// Mitsubishi GX Works2 project: PLC_GROUP2_Final   PLC: FX3G

// global labels: Global1
VAR_GLOBAL
  StartDay AT X007 : BOOL;
  StartRaspberryStock AT D1101 : REAL;
  StartLemonStock AT D1103 : REAL;
  StartStabilizerStock AT D1105 : REAL;
  StartGummyBearsStock AT D1107 : REAL;
  StockRaspberry AT D1111 : REAL;
  LemonStock AT D1133 : REAL;
  RaspberryStock AT D1111 : REAL;
  StabilizerStock AT D1155 : REAL;
  GummyBearsStock AT D1177 : REAL;
  WorkDayLight AT Y007 : BOOL;
  LackOfStock AT M0 : BOOL;
  EmergencySwitch AT X005 : BOOL;
  WorkDayLigth AT Y007 : BOOL;
  IceCreamFlavors AT X001 : BOOL;
  AnalogInput1 AT D8280 : INT;
  SaveAnalogInput1 AT D8201 : INT;
  Analog1AsFloat AT D1221 : REAL;
  Divider AT E400 : REAL;
  IndicatorLigth AT M1 : BOOL;
  RegularLigth AT M2 : BOOL;
  IndulgenceLigth AT M3 : BOOL;
  CheckStock AT M100 : BOOL;
END_VAR
VAR_GLOBAL CONSTANT
  RaspberryForPackage : REAL := 280;
END_VAR
VAR_GLOBAL
  RegularPackage AT M22 : BOOL;
END_VAR
VAR_GLOBAL CONSTANT
  Regular : REAL := 5;
END_VAR
VAR_GLOBAL
  RegularCheck AT M2 : BOOL;
  IndulgencePackage AT M33 : BOOL;
END_VAR
VAR_GLOBAL CONSTANT
  Indulgence : INT := 6;
  IndulgenceMin : REAL := 6;
  LemonForPackage : REAL := 455;
  StabilizerForPackage : REAL := 105;
  GummyBearsForPackage : REAL := 28;
  RaspberryForPackage3 : REAL := 385;
  LemonForPackage3 : REAL := 665;
  StabilizerForPackage3 : REAL := 210;
  GummyBearsForPackage3 : REAL := 70;
  RaspberryForPackage2 : INT := 280;
  GummyBearsForPackage2 : INT := 280;
  addRaspberry : REAL := 350;
  addLemon : REAL := 490;
  addRaspberry3 : REAL := 560;
  addLemon3 : REAL := 700;
END_VAR
VAR_GLOBAL
  FlavorsMaking AT M40 : BOOL;
END_VAR
VAR_GLOBAL CONSTANT
  TotIceCreamTime : INT := 50;
END_VAR
VAR_GLOBAL
  IceCreamTime AT TC1 : BOOL;
  MakingTime AT Y000 : BOOL;
  MakingTimer AT TS1 : BOOL;
  Cooling AT X002 : BOOL;
  TemperatureSensor AT X003 : BOOL;
END_VAR
VAR_GLOBAL CONSTANT
  MaxTime : INT := 80;
END_VAR
VAR_GLOBAL
  CoolingTime AT TC8 : BOOL;
  CoolingTimer AT TS8 : BOOL;
  CoolingLight AT Y002 : BOOL;
END_VAR
VAR_GLOBAL CONSTANT
  GummyBearskForPackage : REAL := 28;
  GummyBearskForPackage3 : REAL := 70;
END_VAR
VAR_GLOBAL
  RegularMix AT M4 : BOOL;
  IndulgenceMix AT M5 : BOOL;
END_VAR
VAR_GLOBAL CONSTANT
  RegularMix3sec : INT := 30;
  IndulgenceMix5sec : INT := 50;
END_VAR
VAR_GLOBAL
  StartMix AT M4 : BOOL;
  LightTimer AT TS9 : BOOL;
  LightTime AT TC9 : BOOL;
  FirstLight AT Y005 : BOOL;
  SecondLight AT Y006 : BOOL;
  HelpLight AT M5 : BOOL;
  FirstLightTime AT TC10 : BOOL;
  SecondLightTime AT TC11 : BOOL;
  FirstLightTimer AT TS10 : BOOL;
  SecondLightTimer AT TS11 : BOOL;
  IndulgenceChecking AT M6 : BOOL;
  CoolingRaspberry AT D2004 : REAL;
  CoolingLemon AT D2006 : REAL;
  MixingFlavors AT D3000 : REAL;
END_VAR
VAR_GLOBAL CONSTANT
  Restart : INT;
END_VAR
VAR_GLOBAL
  AnalogOutput AT D8282 : INT;
  RaspberryIceCream AT D2000 : REAL;
  LemonIceCream AT D2002 : REAL;
  Checking AT Y010 : BOOL;
  ch AT Y011 : BOOL;
  StayOn AT M50 : BOOL;
  Help AT M50 : BOOL;
  FlavorsMaking12 AT M42 : BOOL;
  HelpCooling AT M60 : BOOL;
  MixTimerWord AT D3006 : INT;
  MixTimer AT D3002 : REAL;
END_VAR
VAR_GLOBAL CONSTANT
  MaxTime2 : INT := 8;
END_VAR
VAR_GLOBAL
  LightTime3 AT TC12 : BOOL;
  LightTimer3 AT TS12 : BOOL;
  Help7 AT M7 : BOOL;
  Check4 AT Y010 : BOOL;
  Check10 AT Y004 : BOOL;
  Packing AT X004 : BOOL;
END_VAR
VAR_GLOBAL CONSTANT
  RstMixingFlavors : REAL;
END_VAR
VAR_GLOBAL
  OneCone AT X000 : BOOL;
  FirstConeCounter AT CC0 : BOOL;
END_VAR
VAR_GLOBAL CONSTANT
  FirstCone : INT := 1;
END_VAR
VAR_GLOBAL
  ConesCounter AT CC1 : BOOL;
END_VAR
VAR_GLOBAL CONSTANT
  SevenCones : INT := 7;
END_VAR
VAR_GLOBAL
  AfterFirstCone AT CS0 : BOOL;
  FinishPackeg AT CS1 : BOOL;
  FinishPackage AT CS1 : BOOL;
  PackingLigth AT Y004 : BOOL;
END_VAR
VAR_GLOBAL CONSTANT
  NewPackage : REAL := 1;
END_VAR
VAR_GLOBAL
  TotalPackages AT D5555 : REAL;
END_VAR
VAR_GLOBAL CONSTANT
  Mult : REAL := 40;
  Reset : REAL;
END_VAR
VAR_GLOBAL
  StartReset AT M8 : BOOL;
  HelpM41 AT M41 : BOOL;
  closeLigth AT M100 : BOOL;
END_VAR

// task Task_01 (event TRUE, interval 0, priority 31): POU_01

PROGRAM POU_01
(* structured ladder/FBD written out as ST: instructions are called as NAME(EN, inputs, outputs); _pN, _eN, _tN stand for wires *)
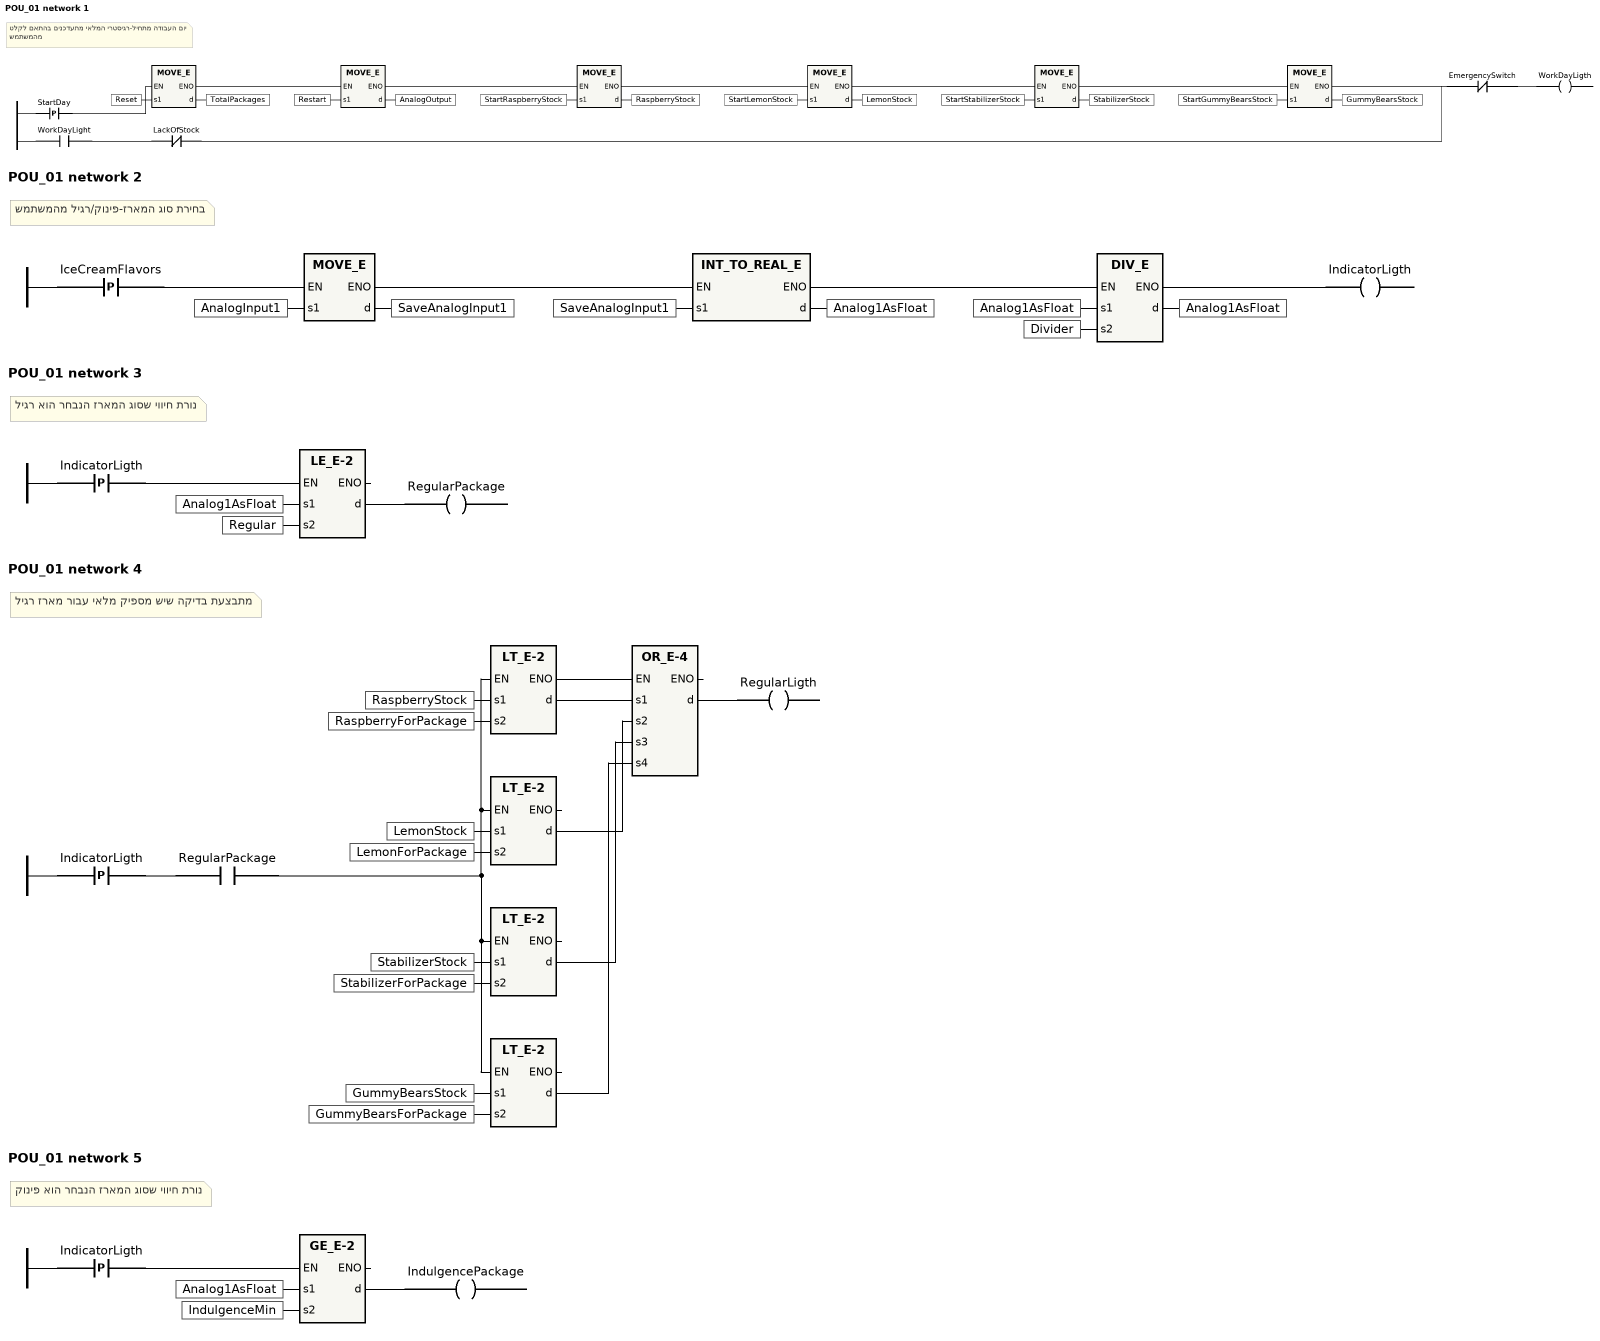
(* network 1 Start workday *)
(* יום העבודה מתחיל-רגיסטרי המלאי מתעדכנים בהתאם לקלט מהמשתמש *)
_e1 := MOVE_E(LDP(TRUE, StartDay), Reset, TotalPackages);
_e2 := MOVE_E(_e1, Restart, AnalogOutput);
_e3 := MOVE_E(_e2, StartRaspberryStock, RaspberryStock);
_e4 := MOVE_E(_e3, StartLemonStock, LemonStock);
_e5 := MOVE_E(_e4, StartStabilizerStock, StabilizerStock);
_e6 := MOVE_E(_e5, StartGummyBearsStock, GummyBearsStock);
WorkDayLigth := (_e6 OR (WorkDayLight AND NOT LackOfStock)) AND NOT EmergencySwitch;
(* network 2 Type sampeling *)
(* בחירת סוג המארז-פינוק/רגיל מהמשתמש *)
_e1 := MOVE_E(LDP(TRUE, IceCreamFlavors), AnalogInput1, SaveAnalogInput1);
_e2 := INT_TO_REAL_E(_e1, SaveAnalogInput1, Analog1AsFloat);
_e3 := DIV_E(_e2, Analog1AsFloat, Divider, Analog1AsFloat);
IndicatorLigth := _e3;
(* network 3 If regular *)
(* נורת חיווי שסוג המארז הנבחר הוא רגיל *)
LE_E(LDP(TRUE, IndicatorLigth), Analog1AsFloat, Regular, _t1);
RegularPackage := _t1;
(* network 4 Check stock for R *)
(* מתבצעת בדיקה שיש מספיק מלאי עבור מארז רגיל *)
_p1 := LDP(TRUE, IndicatorLigth) AND RegularPackage;
_e3 := LT_E(_p1, RaspberryStock, RaspberryForPackage, _t2);
LT_E(_p1, LemonStock, LemonForPackage, _t4);
LT_E(_p1, StabilizerStock, StabilizerForPackage, _t5);
LT_E(_p1, GummyBearsStock, GummyBearsForPackage, _t6);
OR_E(_e3, _t2, _t4, _t5, _t6, _t7);
RegularLigth := _t7;
(* network 5 If indulgence *)
(* נורת חיווי שסוג המארז הנבחר הוא פינוק *)
GE_E(LDP(TRUE, IndicatorLigth), Analog1AsFloat, IndulgenceMin, _t1);
IndulgencePackage := _t1;
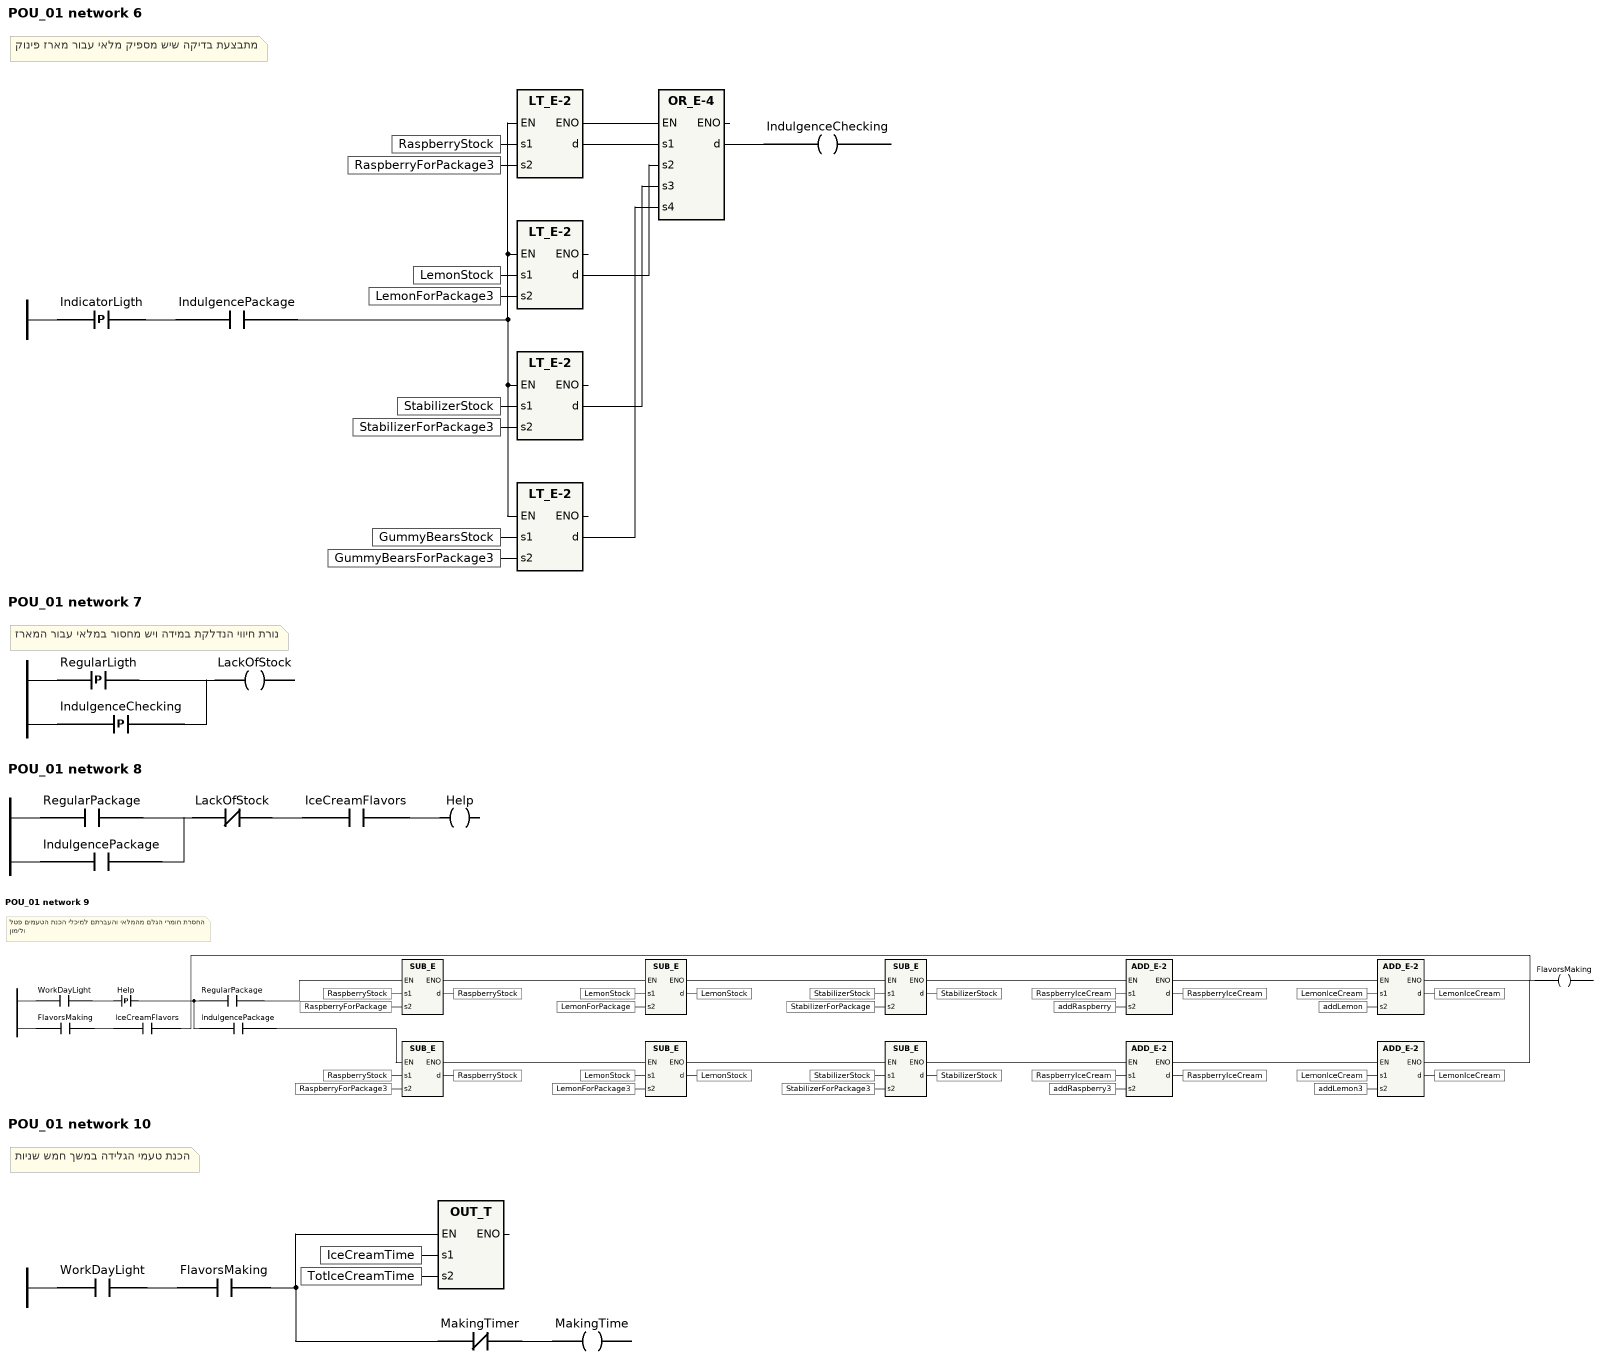
(* network 6 Check stock for I *)
(* מתבצעת בדיקה שיש מספיק מלאי עבור מארז פינוק *)
_p1 := LDP(TRUE, IndicatorLigth) AND IndulgencePackage;
_e3 := LT_E(_p1, RaspberryStock, RaspberryForPackage3, _t2);
LT_E(_p1, LemonStock, LemonForPackage3, _t4);
LT_E(_p1, StabilizerStock, StabilizerForPackage3, _t5);
LT_E(_p1, GummyBearsStock, GummyBearsForPackage3, _t6);
OR_E(_e3, _t2, _t4, _t5, _t6, _t7);
IndulgenceChecking := _t7;
(* network 7 Out of stock *)
(* נורת חיווי הנדלקת במידה ויש מחסור במלאי עבור המארז *)
LackOfStock := LDP(TRUE, RegularLigth) OR LDP(TRUE, IndulgenceChecking);
(* network 8 Checks conditions *)
Help := ((RegularPackage OR IndulgencePackage) AND NOT LackOfStock) AND IceCreamFlavors;
(* network 9 Sub stocks *)
(* החסרת חומרי הגלם מהמלאי והעברתם למיכלי הכנת הטעמים פטל ולימון *)
_p1 := WorkDayLight AND LDP(TRUE, Help);
_e2 := SUB_E(_p1 AND RegularPackage, RaspberryStock, RaspberryForPackage, RaspberryStock);
_e3 := SUB_E(_e2, LemonStock, LemonForPackage, LemonStock);
_e4 := SUB_E(_e3, StabilizerStock, StabilizerForPackage, StabilizerStock);
_e5 := ADD_E(_e4, RaspberryIceCream, addRaspberry, RaspberryIceCream);
_e6 := ADD_E(_e5, LemonIceCream, addLemon, LemonIceCream);
_e7 := SUB_E(_p1 AND IndulgencePackage, RaspberryStock, RaspberryForPackage3, RaspberryStock);
_e8 := SUB_E(_e7, LemonStock, LemonForPackage3, LemonStock);
_e9 := SUB_E(_e8, StabilizerStock, StabilizerForPackage3, StabilizerStock);
_e10 := ADD_E(_e9, RaspberryIceCream, addRaspberry3, RaspberryIceCream);
_e11 := ADD_E(_e10, LemonIceCream, addLemon3, LemonIceCream);
FlavorsMaking := _e6 OR _e11 OR (FlavorsMaking AND IceCreamFlavors);
(* network 10 Flavors Making *)
(* הכנת טעמי הגלידה במשך חמש שניות *)
_p1 := WorkDayLight AND FlavorsMaking;
OUT_T(_p1, IceCreamTime, TotIceCreamTime);
MakingTime := _p1 AND NOT MakingTimer;
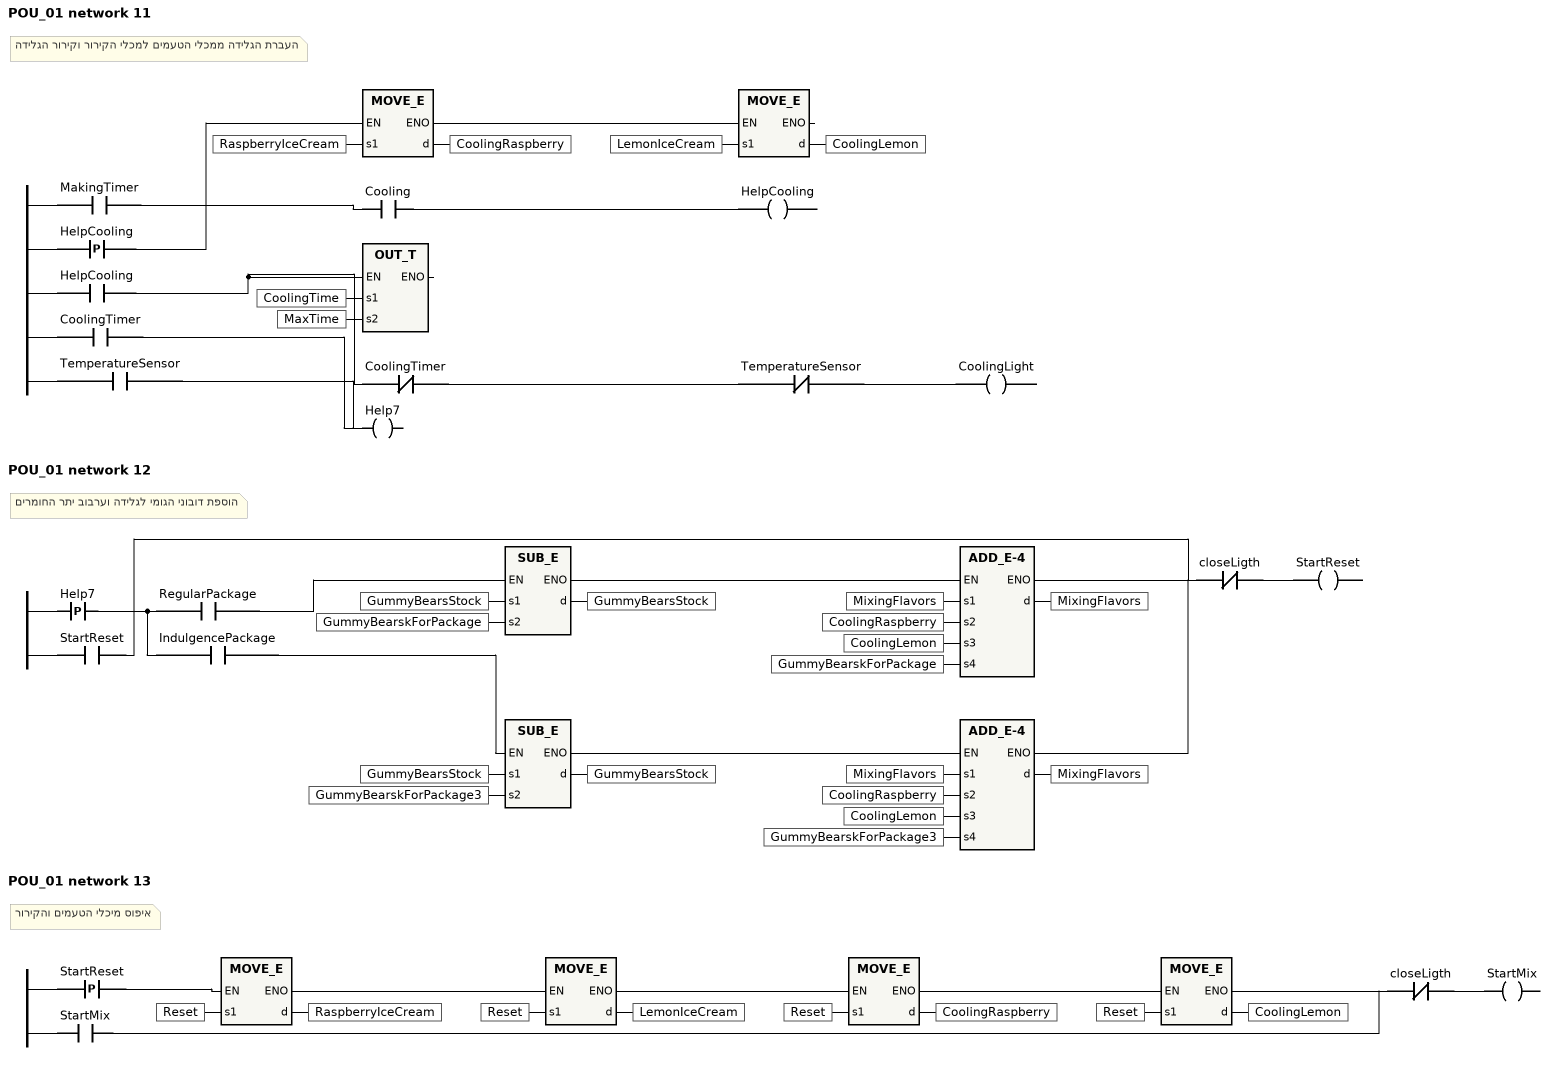
(* network 11 Cooling phase *)
(* העברת הגלידה ממכלי הטעמים למכלי הקירור וקירור הגלידה *)
HelpCooling := MakingTimer AND Cooling;
_e1 := MOVE_E(LDP(TRUE, HelpCooling), RaspberryIceCream, CoolingRaspberry);
MOVE_E(_e1, LemonIceCream, CoolingLemon);
OUT_T(HelpCooling, CoolingTime, MaxTime);
CoolingLight := HelpCooling AND NOT CoolingTimer AND NOT TemperatureSensor;
Help7 := CoolingTimer OR TemperatureSensor;
(* network 12 Prepar to Mixing *)
(* הוספת דובוני הגומי לגלידה וערבוב יתר החומרים *)
_p1 := LDP(TRUE, Help7);
_e2 := SUB_E(_p1 AND RegularPackage, GummyBearsStock, GummyBearskForPackage, GummyBearsStock);
_e3 := ADD_E(_e2, MixingFlavors, CoolingRaspberry, CoolingLemon, GummyBearskForPackage, MixingFlavors);
_e4 := SUB_E(_p1 AND IndulgencePackage, GummyBearsStock, GummyBearskForPackage3, GummyBearsStock);
_e5 := ADD_E(_e4, MixingFlavors, CoolingRaspberry, CoolingLemon, GummyBearskForPackage3, MixingFlavors);
StartReset := (_e3 OR _e5 OR StartReset) AND NOT closeLigth;
(* network 13 Restart *)
(* איפוס מיכלי הטעמים והקירור *)
_e1 := MOVE_E(LDP(TRUE, StartReset), Reset, RaspberryIceCream);
_e2 := MOVE_E(_e1, Reset, LemonIceCream);
_e3 := MOVE_E(_e2, Reset, CoolingRaspberry);
_e4 := MOVE_E(_e3, Reset, CoolingLemon);
StartMix := (_e4 OR StartMix) AND NOT closeLigth;
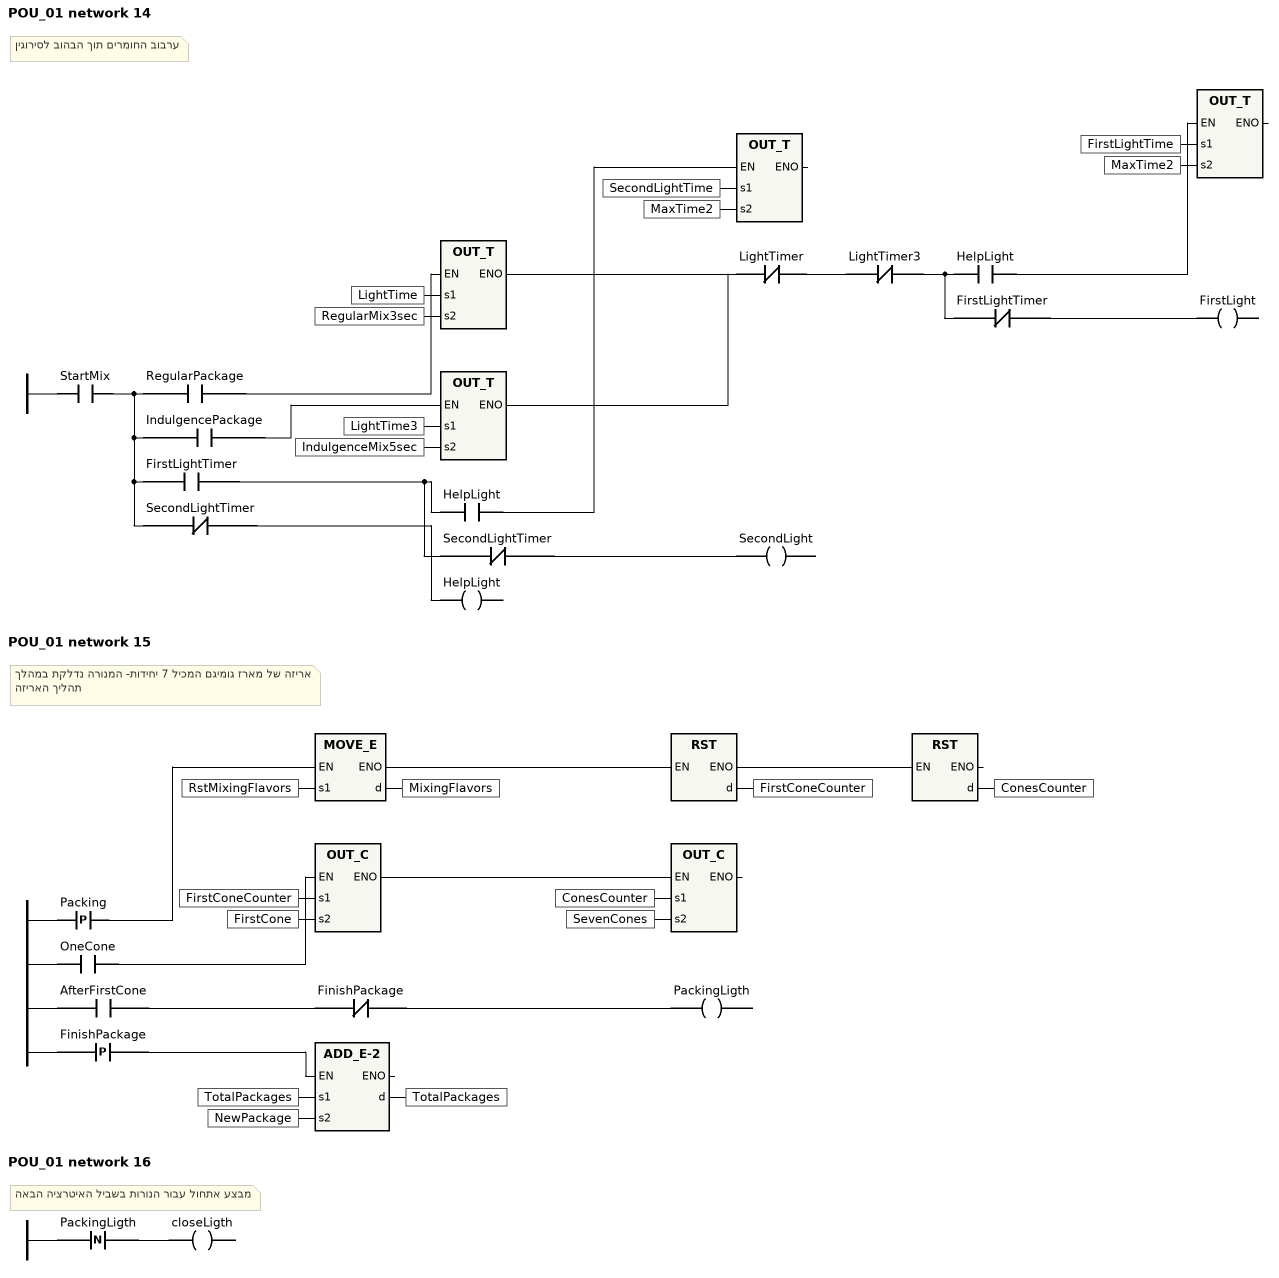
(* network 14 Mixing Ingredients *)
(* ערבוב החומרים תוך הבהוב לסירוגין *)
_e1 := OUT_T(StartMix AND RegularPackage, LightTime, RegularMix3sec);
_e2 := OUT_T(StartMix AND IndulgencePackage, LightTime3, IndulgenceMix5sec);
_p3 := ((_e1 OR _e2) AND NOT LightTimer) AND NOT LightTimer3;
OUT_T(_p3 AND HelpLight, FirstLightTime, MaxTime2);
FirstLight := _p3 AND NOT FirstLightTimer;
_p4 := StartMix AND FirstLightTimer;
OUT_T(_p4 AND HelpLight, SecondLightTime, MaxTime2);
SecondLight := _p4 AND NOT SecondLightTimer;
HelpLight := StartMix AND NOT SecondLightTimer;
(* network 15 Packing cones *)
(* אריזה של מארז גומיגם המכיל 7 יחידות- המנורה נדלקת במהלך תהליך האריזה *)
_e1 := MOVE_E(LDP(TRUE, Packing), RstMixingFlavors, MixingFlavors);
_e2 := RST(_e1, FirstConeCounter);
RST(_e2, ConesCounter);
_e3 := OUT_C(OneCone, FirstConeCounter, FirstCone);
OUT_C(_e3, ConesCounter, SevenCones);
PackingLigth := AfterFirstCone AND NOT FinishPackage;
ADD_E(LDP(TRUE, FinishPackage), TotalPackages, NewPackage, TotalPackages);
(* network 16 Restart bulbs *)
(* מבצע אתחול עבור הנורות בשביל האיטרציה הבאה *)
closeLigth := LDF(TRUE, PackingLigth);
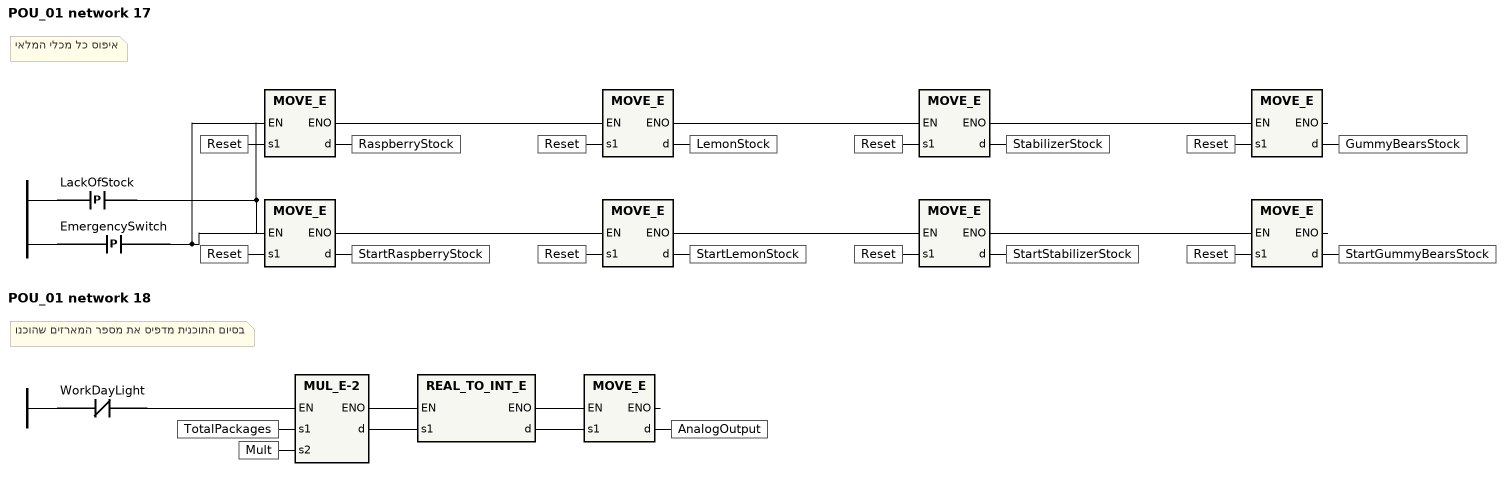
(* network 17 Reset stock *)
(* איפוס כל מכלי המלאי *)
_p1 := LDP(TRUE, LackOfStock) OR LDP(TRUE, EmergencySwitch);
_e2 := MOVE_E(_p1, Reset, RaspberryStock);
_e3 := MOVE_E(_e2, Reset, LemonStock);
_e4 := MOVE_E(_e3, Reset, StabilizerStock);
MOVE_E(_e4, Reset, GummyBearsStock);
_e5 := MOVE_E(_p1, Reset, StartRaspberryStock);
_e6 := MOVE_E(_e5, Reset, StartLemonStock);
_e7 := MOVE_E(_e6, Reset, StartStabilizerStock);
MOVE_E(_e7, Reset, StartGummyBearsStock);
(* network 18 Packages output *)
(* בסיום התוכנית מדפיס את מספר המארזים שהוכנו *)
_e2 := MUL_E(NOT WorkDayLight, TotalPackages, Mult, _t1);
_e4 := REAL_TO_INT_E(_e2, _t1, _t3);
MOVE_E(_e4, _t3, AnalogOutput);
END_PROGRAM
